// TwinCAT 3 PLC project MOTOR_TESTI
// ProgramVersion: 3.1.4024.0
// libraries:
//   Tc2_ControllerToolbox, * (Beckhoff Automation GmbH)
//   Tc2_EtherCAT, * (Beckhoff Automation GmbH)
//   Tc2_MC2, * (Beckhoff Automation GmbH)
//   Tc2_Standard, * (Beckhoff Automation GmbH)
//   Tc2_System, * (Beckhoff Automation GmbH)
//   Tc3_Module, * (Beckhoff Automation GmbH)
// project tree:
//   GVLs/ MAIN_GVL.TcGVL
//   / PlcTask.TcTTO
//   POUs/ COE_READ_WRITE.TcPOU, MAIN.TcPOU, SINGEN.TcPOU
// real-time tasks:
//   TASK PlcTask: cycle T#10ms, priority 20, ADS port 350
// motion (NC):
//   TASK NC-Task 1 SAF: cycle T#10ms, priority 4, ADS port 501
//   TASK NC-Task 1 SVB: cycle T#10ms, priority 8, ADS port 511
//   AXIS Axis 1 (id 1)
//     General: UnitName=°
//     Velo: Maximum=9600
//     OtherSettings: AllowMotionCmdToSlave=true
//     encoder EncType=19
//       EncPara: ScaleFactorNumerator=0.087890625, MaxCount=#xffffffff
//     drive DrvType=16
//       DrvPara: MaxCount=#xffffffff
//         Analog: VeloReferenz=9600, TorqueSetpointScale=10, ScaleFactorActTorque=0.1
//         TimeComp: TaskDelayCycles=1
//     controller CtrType=1
//       CtrPara: PriorControlFactor=1
//         PosDiffControl: Enable=false
//         Observer: BandWidth=20
// I/O:
//   DEVICE Device 5 (EtherCAT), AmsNetId 192.168.137.220.6.1
//     Term 1 (EK1100) [EK1100 EtherCAT Coupler (2A E-Bus)]
//       Term 2 (EL3004) [EL3004 4Ch. Ana. Input +/-10V]
//       Term 3 (EL3218) [EL3218-0000 8Ch. Ana. Input PT100 (RTD)]
//       Term 4 (EL1809) [EL1809 16Ch. Dig. Input 24V, 3ms]
//       Term 5 (EL2809) [EL2809 16Ch. Dig. Output 24V, 0.5A]
//       Term 7 (EL9011) [EL9011 End Terminal]
//     Drive 6 (
            HiDrive
        ) [HiDrive - EtherCAT (CoE) - Profile: Basic & Object Dictionary (v.7.0)]
// variable links:
//   NC-Task 1 SAF/Axes/Axis 1 <-> Device 5 (EtherCAT)/Drive 6 (
            HiDrive
        )
//     Drive/Inputs/In/nState1 <-> Tx PDO4/Status Word
//     Drive/Inputs/In/nState2 <-> Tx PDO4/Status Word @bit 8
//     Drive/Inputs/In/nState4 @bit 1 <-> WcState/InputToggle
//     Drive/Inputs/In/nState4 <-> WcState/WcState
//     Drive/Outputs/Out/nCtrl1 <-> Rx PDO4/Control Word
//     Drive/Outputs/Out/nCtrl2 <-> Rx PDO4/Control Word @bit 8
//     Enc/Inputs/In/nDataIn1 <-> Tx PDO4/Position Actual Value
//     Enc/Inputs/In/nState4 @bit 1 <-> WcState/InputToggle
//     Enc/Inputs/In/nState4 <-> WcState/WcState
//   MOTOR_TESTI/MOTOR_TESTI Instance <-> Device 5 (EtherCAT)/Drive 6 (
            HiDrive
        )
//     PlcTask Inputs/MAIN.OPERATING_MODE_1_READ <-> Tx PDO3/Pr[181] - Operating Mode
//     PlcTask Inputs/MAIN.TORQUE_MONITOR_1 <-> Tx PDO3/Pr[35] - Torque Monitor [0.1% Ipeak]
//     PlcTask Inputs/MAIN.WINDING_THERMAL_IMAGE <-> Tx PDO3/Pr[36] - Winding Thermal Image [0.1%]
//     PlcTask Outputs/MAIN.HIDRIVE_PLC_OUT_1 <-> Rx PDO4/Target Position
//     PlcTask Outputs/MAIN.OPERATING_MODE_1_WRITE <-> Rx PDO3/Pr[181] - Operating Mode
//     PlcTask Outputs/SINGEN.PR5_INTERNALSETPOINT_1 <-> Rx PDO3/Pr[5] - Internal SetPoint [rpm]
//   MOTOR_TESTI/MOTOR_TESTI Instance <-> Device 5 (EtherCAT)/Term 1 (EK1100)/Term 2 (EL3004)
//     PlcTask Inputs/MAIN.TEST_TORQUE_SENSOR_1 <-> AI Standard Channel 3/Value
//     PlcTask Inputs/MAIN.VOL_READ_1 <-> AI Standard Channel 1/Value
//     PlcTask Inputs/MAIN.VOL_READ_2 <-> AI Standard Channel 2/Value
//   MOTOR_TESTI/MOTOR_TESTI Instance <-> NC-Task 1 SAF/Axes/Axis 1
//     PlcTask Inputs/MAIN.HIDRIVE_PLC_IN_1 <-> Drive/Outputs/Out/nDataOut1
//     PlcTask Inputs/MAIN_GVL.MOTOR_AXIS1.NcToPlc <-> Outputs/ToPlc
//     PlcTask Outputs/MAIN_GVL.MOTOR_AXIS1.PlcToNc <-> Inputs/FromPlc

CONFIGURATION MOTOR_TESTI
    RESOURCE PLC ON TwinCAT3
        TASK PlcTask(INTERVAL := T#10ms, PRIORITY := 20);
        PROGRAM MAIN WITH PlcTask : MAIN;
    END_RESOURCE
END_CONFIGURATION

// ---- GVLs/MAIN_GVL.TcGVL
{attribute 'qualified_only'}
VAR_GLOBAL
	
	MC_POWER_MOTOR: MC_POWER;
	MOTOR_AXIS1: AXIS_REF;
	
	ENABLE_MOTOR: BOOL;
	OverrideRatio: REAL:=100;
END_VAR

// ---- POUs/MAIN.TcPOU
PROGRAM MAIN
VAR
	HIDRIVE_PLC_IN_1 AT%I* : DINT; // MOTION/DRIVE İÇİNDE / OUTPUT / NDATAOUT1 LİNKİNE EKLENİR
	HIDRIVE_PLC_OUT_1 AT%Q* : DINT; // HIDRIVE İÇİNDE RX PDO4 İÇİNDEKİ TARGET POSİTİONA LİNKLENİR BU LİNKLEME YAPILMAZSA MOTOR ÇALIŞMAZ
	TORQUE_MONITOR_1 AT%I* : INT ;
	CURRENT_ACTUAL : REAL;
	MAX_PEEK_CURRENT : INT := 10;
	
	OPERATING_MODE_1_WRITE AT%Q* : INT:=203; // 0 SPEED CONTROL - 203 ETHERCAT - 110 CURRENT
		OPERATING_MODE_1_READ AT%I* : INT; // 0 SPEED CONTROL - 203 ETHERCAT - 110 CURRENT
		OPERATING_MODE_1_READ_SCADA: REAL;
		//ug
		WINDING_THERMAL_IMAGE AT %I* : INT;
	OPMODE_CHANGE: BOOL;
	OPMODE: REAL;
	VOL_READ_1 AT %I* : INT ;
	VOL_READ_2 AT %I* : INT ;
	TORQ_VOLTAGE_HESAP : REAL;
	TORQ_VOLTAGE_OFFSET : REAL := 2.63;
	TORQ_VOLTAGE_FARK : REAL;
	A : LREAL := -3.00499219E-02;
	B : LREAL := 1.73472887E-02;
	C : LREAL := 9.69692536E+00;
	TORQ_ACTUAL : LREAL;
	
	M_TORQ : REAL := 9.2348; // 9.2348
	N_TORQ : REAL := -24.057; // -24.057
	TEST_TORQUE_SENSOR_1 AT %I* : INT ;
	M_TEST : INT := 409;
	N_TEST : INT := 204;
	KISSLER_TORQUE_SENSOR_SCALED: REAL;

	REVOLUTION_RadSn : REAL;
	REVOLUTION_RPM: LREAL; //FROM BECKHOFF NC ( NUMERIC/Motion CONTROL )
	
	Torque_Offset : REAL;
	
	
//	bStartScope : BOOL;
//	bStopScope : BOOL;
//	bExportScope : BOOL;
//	Kontrol1: BOOL;
//	Kontrol2: BOOL;
//	Kontrol3: BOOL;
	
//	SET_TO_SETPOINT2 : INT;
	
//	StartCase: BOOL;
//	RestartCase: BOOL;
	
//	fbTimer: TON;
//	bTriggerTimer1: BOOL;
//	bTriggerTimer2: BOOL;
//	bTriggerTimer3: BOOL;

//	nState: UDINT := 0;
	
	eReqState	:BOOL;
	
END_VAR

REVOLUTION_RPM:=(Main_Gvl.MOTOR_AXIS1.NcToPlc.ActVelo/360)*60;
CURRENT_ACTUAL := INT_TO_REAL(TORQUE_MONITOR_1) * MAX_PEEK_CURRENT / 1000;
IF HIDRIVE_PLC_OUT_1=0 THEN
	MAIN_GVL.ENABLE_MOTOR:=FALSE;
END_IF
HIDRIVE_PLC_OUT_1 := HIDRIVE_PLC_IN_1;
OPERATING_MODE_1_READ_SCADA:=INT_TO_REAL(OPERATING_MODE_1_READ);
IF OPMODE_CHANGE THEN
	OPERATING_MODE_1_WRITE:=REAL_TO_INT(OPMODE);
	OPMODE_CHANGE:=FALSE;
END_IF

//TORQ_HESAP_1 := M_TORQ*((VOL_READ_1/32768)*10) - N_TORQ;
TORQ_VOLTAGE_HESAP := INT_TO_REAL(VOL_READ_1)/32768 *10;

TORQ_VOLTAGE_FARK := TORQ_VOLTAGE_HESAP - TORQ_VOLTAGE_OFFSET;
TORQ_ACTUAL := A*(TORQ_VOLTAGE_FARK*TORQ_VOLTAGE_FARK*TORQ_VOLTAGE_FARK) + B*(TORQ_VOLTAGE_FARK*TORQ_VOLTAGE_FARK) + C*TORQ_VOLTAGE_FARK;


REVOLUTION_RadSn := REVOLUTION_RPM*2*3.14159/60;

KISSLER_TORQUE_SENSOR_SCALED:=((INT_TO_REAL(VOL_READ_1)-8192)/6554)*17.5;

MAIN_GVL.MC_POWER_MOTOR(
	Axis:=MAIN_GVL.MOTOR_AXIS1 , 
	Enable:=MAIN_GVL.ENABLE_MOTOR , 
	Enable_Positive:=MAIN_GVL.ENABLE_MOTOR , 
	Enable_Negative:=MAIN_GVL.ENABLE_MOTOR , 
	Override:=MAIN_GVL.OverrideRatio, 
	BufferMode:= , 
	Options:= , 
	Status=> , 
	Busy=> , 
	Active=> , 
	Error=> , 
	ErrorID=> );
	

	
	
	COE_READ_WRITE();
	SINGEN();

END_PROGRAM

// ---- POUs/COE_READ_WRITE.TcPOU
PROGRAM COE_READ_WRITE
VAR
coe_write          : FB_EcCoESdoWrite; // Function Block for writing in CoE
   coe_read           : FB_EcCoESdoRead;  // Function Block for reading from CoE
   userNetId             : T_AmsNetId := '5.94.222.87.1.1'; // Have to be entered
   userSlaveAddr         : UINT := 1006;     // Have to be entered
   startWrite            : BOOL := FALSE;    // Sign for start writing
   startRead             : BOOL := FALSE;    // Sign for start reading
   nState                : BYTE := 0;        // RW-status
   // Example: Read EL3751 PAI Internal Data: Temperature Value
   int16Buffer           : INT;              // Buffer for reading
   // Example: Select EL3751 Filter1: 22 = IIR Butterw. LP 5th Ord. 1000 Hz:
   uint16Buffer          : UINT:=22;         // Buffer for writing
   bTxPDOState AT%I*     : BOOL;             // (PDO for synchronization)
	EXEC: BOOL;
	bBusy: STRING(INT#4);
	EXEC_wRITE: BOOL;
END_VAR


coe_read(
   sNetId:= '5.94.222.87.1.1', 
   nSlaveAddr:= userSlaveAddr, 
   nSubIndex:= 16#11, 
   nIndex:= 16#2000,
   pDstBuf:= ADR(int16Buffer), 
   cbBufLen:= 16, 
   bExecute:= EXEC, 
   tTimeout:= T#1S,
   );
    // Write entry
   coe_write(
   sNetId:= userNetId,
   nSlaveAddr:= userSlaveAddr,
   nSubIndex:= 16#11,
   nIndex:= 16#2000,
   pSrcBuf:= ADR(uint16Buffer),
   cbBufLen:= 2,
   bExecute:= EXEC_wRITE,
   tTimeout:= T#1S
   );

END_PROGRAM

// ---- POUs/SINGEN.TcPOU
PROGRAM SINGEN
VAR
	DEGREE: INT;
	SINE_MODE_SELECT: REAL;
	SINGEN: FB_CTRL_SIGNAL_GENERATOR;
	SINGEN_SWEEP: FB_CTRL_SIGNAL_GENERATOR;
	State: E_CTRL_STATE;
	ErrorID: E_CTRL_ERRORCODES;
	Error: BOOL;
	WaveOutput: LREAL;
	stParams_deneme: ST_CTRL_SIGNAL_GENERATOR_PARAMS;
	SineSweep_params: ST_CTRL_SIGNAL_GENERATOR_PARAMS;
	Signal_Type: E_CTRL_SIGNAL_TYPE;
	
	SET_TO_SETPOINT: REAL;

	start : BOOL;
	
	eMode_deneme: E_CTRL_MODE;
	SINE_SWEEP: BOOL;
	CLOCK: INT;

	CLOCK_1: INT;
	AT_OFFSET: BOOL;
	SINE_GENERATOR: BOOL;
	
	RPM_TO_Degree_1: LREAL;
	PR5_INTERNALSETPOINT_1 AT%Q*: INT;
	CURRENT_REFERENCE : INT;
	VELOCITY_REFERENCE_rpm : INT;
	VELOCITY_REFERENCE_RadSn : LREAL;
	
	RPM_TO_Degree_2: LREAL;
	PR5_INTERNALSETPOINT_2 AT%Q*: INT;
	
	RPM_TO_Degree_4: LREAL;
	PR5_INTERNALSETPOINT_4 AT%Q*: INT;
	
	RPM_TO_Degree_5: LREAL;
	PR5_INTERNALSETPOINT_5 AT%Q*: INT;
	
	SineWave_PERIOD: TIME:=T#10S;
	SineSweep_PERIOD:TIME:=T#10S;
	MANUAL_SET_POINT: BOOL;
	
	SINE_OFFSET: REAL:=0;
	SINE_AMPLITUDE: REAL:=10;
	CTRL_CYCLE_TIME: TIME:=T#10MS;
	CTRL_TIME_FROM_SCADA: REAL:=10;
	TASK_CYCLE_TIME: TIME:=T#10MS;
	TASK_TIME_FROM_SCADA : REAL:=10;
	PERIOD_FROM_SCADA: REAL:=10;
	
	START_TIME_OFFSET: TIME:=T#0MS;
	START_TIME_FROM_SCADA:REAL;
	
	MAX_SineSweep_PERIOD: TIME := T#1000MS;
	MAX_SineSweep_PERIOD_FROM_SCADA: REAL:=1000;
	SET_SETPOINT_0: BOOL;
	START_SINE: BOOL;
	STOP_SINE: BOOL;
	SCADA_ONLINE: BOOL:=TRUE;
	FB_CTRL_GET_TASK_CYCLETIME: FB_CTRL_GET_TASK_CYCLETIME;
	TaskCycleTime: TIME;
	bCycleTimeValid: BOOL;
	eState: Tc2_ControllerToolbox.E_CTRL_STATE;
	ErrID: Tc2_ControllerToolbox.E_CTRL_ERRORCODES;
	Err: BOOL;
	check1: BOOL;
	FALLDOWN_RATIO: REAL:=2;
	SWEEPPERIOD_FROM_SCADA: REAL;
	ONE_TIME_CHECK: BOOL;
	ONE_TIME_CHECK2: BOOL;
	SinSweep_PERIOD_FOR_SCADA: REAL;
	MAX_SineSweep_PERIOD_FOR_SCADA: REAL;
	START_TIME_OFFSET_FOR_SCADA: REAL;
	TASK_CYCLE_TIME_FOR_SCADA: REAL;
	SineSweep_PERIOD_FOR_SCADA:REAL;
	SineWave_PERIOD_FOR_SCADA:REAL;
	CTRL_CYCLE_TIME_FOR_SCADA:REAL;
	
	torqueValues: ARRAY[0..19] OF REAL := [-150, -120, -100 , -80, -60, -40, -20, -10, -5, -1, 1, 5, 10, 20, 40, 60, 80, 100, 120, 150];
	torqueGain : REAL := 1;
	counter: INT := 0;
	index: INT := 0;
	duration: INT := 500;
	
	bSingenStartScope : BOOL;
	bSingenStopScope : BOOL;
	bSingenExportScope : BOOL;
	
	Kontrol1: BOOL;
	Kontrol2: BOOL;
	Kontrol3: BOOL;
	
	StartCase: BOOL;
	RestartCase: BOOL;
	
	fbTimer1: TON;
	fbTimer2: TON;
	fbTimer3: TON;

	bTriggerTimer1: BOOL;
	bTriggerTimer2: BOOL;
	bTriggerTimer3: BOOL;

	nState: UDINT := 0;
	
END_VAR

CURRENT_REFERENCE := PR5_INTERNALSETPOINT_1;
VELOCITY_REFERENCE_rpm := PR5_INTERNALSETPOINT_1;
VELOCITY_REFERENCE_RadSn := VELOCITY_REFERENCE_rpm*2*3.14159/60;

RPM_TO_Degree_1:= (INT_TO_REAL(PR5_INTERNALSETPOINT_1)/60)*360;
RPM_TO_Degree_2:= (INT_TO_REAL(PR5_INTERNALSETPOINT_2)/60)*360;
RPM_TO_Degree_4:= (INT_TO_REAL(PR5_INTERNALSETPOINT_4)/60)*360;
RPM_TO_Degree_5:= (INT_TO_REAL(PR5_INTERNALSETPOINT_5)/60)*360;


IF counter < duration AND start THEN
	SET_TO_SETPOINT := torqueValues[index]* 9.5493;
	counter := counter + 1;
	IF index > 19 THEN
		SET_TO_SETPOINT := 0;
		index := 0;
		start := FALSE;
	END_IF
	
ELSIF start AND counter >= duration THEN
	index := index +1;
	counter := 0;
END_IF

IF (RestartCase = TRUE) THEN
	nState := 0;	
    bSingenStartScope:=FALSE;
	bSingenStopScope:=FALSE;
	bSingenExportScope:=FALSE;	
	RestartCase := FALSE;
	StartCase := FALSE;
END_IF

CASE nState OF
0:
	IF (StartCase = TRUE) THEN		
		bSingenStartScope:=TRUE;
   	    nState := 10;	
	END_IF

10:
    IF bSingenStartScope THEN
        bTriggerTimer1 := TRUE;
        nState := 20;
    END_IF
20:
    IF (Kontrol1 = TRUE) THEN
        bTriggerTimer1 := FALSE;
		SET_TO_SETPOINT:= 1000;
		PR5_INTERNALSETPOINT_1:=REAL_TO_INT(SET_TO_SETPOINT);
        bTriggerTimer2 := TRUE;
        nState := 30;
    END_IF
30:
    IF (Kontrol2 = TRUE) THEN
        bTriggerTimer2 := FALSE;
		SET_TO_SETPOINT:= 0;
		PR5_INTERNALSETPOINT_1:=REAL_TO_INT(SET_TO_SETPOINT);
        bTriggerTimer3 := TRUE;
        nState := 40;
    END_IF
40: 
    IF (Kontrol3 = TRUE) THEN
        bTriggerTimer3 := FALSE;
		bSingenStopScope := TRUE;
        nState := 50;
    END_IF
50:
    IF bSingenStopScope THEN
        bSingenExportScope:=TRUE;
		//RestartCase := TRUE;

    END_IF
END_CASE

fbTimer1(IN:=bTriggerTimer1, PT:=T#1S, Q=> Kontrol1);	
fbTimer2(IN:=bTriggerTimer2, PT:=T#5S, Q=> Kontrol2);	
fbTimer3(IN:=bTriggerTimer3, PT:=T#1S, Q=> Kontrol3);


IF MANUAL_SET_POINT THEN
	PR5_INTERNALSETPOINT_1:=REAL_TO_INT(SET_TO_SETPOINT);
	PR5_INTERNALSETPOINT_2:=REAL_TO_INT(SET_TO_SETPOINT);
	PR5_INTERNALSETPOINT_4:=REAL_TO_INT(SET_TO_SETPOINT);
	PR5_INTERNALSETPOINT_5:=REAL_TO_INT(SET_TO_SETPOINT);
	IF SET_SETPOINT_0 THEN
	SET_TO_SETPOINT:=0;

	SET_SETPOINT_0:=FALSE;
END_IF



ELSIF NOT MANUAL_SET_POINT AND NOT(SINE_GENERATOR OR SINE_SWEEP) THEN
	PR5_INTERNALSETPOINT_1:=0;
	PR5_INTERNALSETPOINT_2:=0;
	PR5_INTERNALSETPOINT_4:=0;
	PR5_INTERNALSETPOINT_5:=0;
END_IF



IF START_SINE THEN
	eMode_deneme := E_CTRL_MODE.eCTRL_MODE_ACTIVE;
	START_SINE:=FALSE;
	check1:=TRUE;
END_IF

IF STOP_SINE THEN
	eMode_deneme:= e_CTRL_MODE.eCTRL_MODE_PASSIVE;
	STOP_SINE:=FALSE;
END_IF

IF (SINE_GENERATOR AND SINE_SWEEP) OR MANUAL_SET_POINT THEN
	eMode_deneme:=e_CTRL_MODE.eCTRL_MODE_PASSIVE;
END_IF

/// scada tarafından 0 gelirse sinus 1 gelirse saw 2 gelirse triangle
IF SINE_MODE_SELECT=0 THEN
Signal_Type:=E_CTRL_SIGNAL_TYPE.eCTRL_SINUS;
ELSIF SINE_MODE_SELECT=1 THEN
Signal_Type:=E_CTRL_SIGNAL_TYPE.eCTRL_SAWTOOTH;
ELSIF SINE_MODE_SELECT=2 THEN
Signal_Type:=E_CTRL_SIGNAL_TYPE.eCTRL_TRIANGLE;
END_IF

IF SCADA_ONLINE AND NOT (eMode_DENEME= E_CTRL_MODE.eCTRL_MODE_ACTIVE) THEN
CTRL_CYCLE_TIME:=LREAL_TO_TIME(CTRL_TIME_FROM_SCADA);
SineWave_PERIOD:=LREAL_TO_TIME(PERIOD_FROM_SCADA);
SineSweep_PERIOD:=LREAL_TO_TIME(SWEEPPERIOD_FROM_SCADA);
MAX_SineSweep_PERIOD:=REAL_TO_TIME(MAX_SineSweep_PERIOD_FROM_SCADA);
TASK_CYCLE_TIME:=LREAL_TO_TIME(TASK_TIME_FROM_SCADA);
START_TIME_OFFSET:=LREAL_TO_TIME(START_TIME_FROM_SCADA);

END_IF 
IF SINE_GENERATOR THEN
	//SINE Dalgasıın parametreleri, gerekli bilgi infosys de bulunabilir.
	stParams_deneme.eSignalType:=Signal_TYPE;
	stParams_deneme.fAmplitude:=SINE_AMPLITUDE;
	stParams_deneme.tCtrlCycleTime:=CTRL_CYCLE_TIME;
	stParams_deneme.tCylceDuration:=SineWave_PERIOD  ;
	stParams_deneme.tStart:=START_TIME_OFFSET;
	stParams_deneme.tTaskCycleTime:=TASK_CYCLE_TIME;
	stParams_deneme.fOffset:=SINE_OFFSET;
	
	IF eMode_deneme = E_CTRL_MODE.eCTRL_MODE_RESET THEN
		SINGEN(
		fManValue:=, 
		eMode:=eMode_deneme, 
		fOut=> WaveOutput, 
		eState=> State, 
		eErrorId=> ErrorID, 
		bError=> Error, 
		stParams:= SineSweep_params);
	END_IF
	
	IF eMode_deneme = E_CTRL_MODE.eCTRL_MODE_ACTIVE AND AT_OFFSET THEN
		SINGEN(
			fManValue:=, 
			eMode:=eMode_deneme, 
			fOut=> WaveOutput, 
			eState=> State, 
			eErrorId=> ErrorID, 
			bError=> Error, 
			stParams:= stParams_deneme);
		END_IF
		IF eMode_deneme = E_CTRL_MODE.eCTRL_MODE_ACTIVE AND AT_OFFSET THEN
			SET_TO_SETPOINT:=WaveOutput;
			PR5_INTERNALSETPOINT_1:=REAL_TO_INT(SET_TO_SETPOINT);
			PR5_INTERNALSETPOINT_2:=REAL_TO_INT(SET_TO_SETPOINT);
			PR5_INTERNALSETPOINT_4:=REAL_TO_INT(SET_TO_SETPOINT);
			PR5_INTERNALSETPOINT_5:=REAL_TO_INT(SET_TO_SETPOINT);
		END_IF
	END_IF

IF SINE_SWEEP THEN
	//SINE Dalgasıın parametreleri, gerekli bilgi infosys de bulunabilir.
	SineSweep_params.eSignalType:=Signal_TYPE;
	SineSweep_params.fAmplitude:=SINE_AMPLITUDE;
	SineSweep_params.tCtrlCycleTime:=T#10MS;
	SineSweep_params.tCylceDuration:=SineSweep_PERIOD ;
	SineSweep_params.tStart:=T#0MS;
	SineSweep_params.tTaskCycleTime:=T#10MS;
	SineSweep_params.fOffset:=SINE_OFFSET;
	IF eMode_deneme = E_CTRL_MODE.eCTRL_MODE_RESET THEN
		SINGEN_SWEEP(
		fManValue:=, 
		eMode:=eMode_deneme, 
		fOut=> WaveOutput, 
		eState=> State, 
		eErrorId=> ErrorID, 
		bError=> Error, 
		stParams:= SineSweep_params);
	END_IF
	IF eMode_deneme = E_CTRL_MODE.eCTRL_MODE_ACTIVE AND AT_OFFSET THEN
		
		SINGEN_SWEEP(
		fManValue:=, 
		eMode:=eMode_deneme, 
		fOut=> WaveOutput, 
		eState=> State, 
		eErrorId=> ErrorID, 
		bError=> Error, 
		stParams:= SineSweep_params);
		
		IF eMode_deneme = E_CTRL_MODE.eCTRL_MODE_ACTIVE AND AT_OFFSET THEN
			SET_TO_SETPOINT:=LREAL_TO_INT(WaveOutput);
			PR5_INTERNALSETPOINT_1:=REAL_TO_INT(SET_TO_SETPOINT);
			PR5_INTERNALSETPOINT_2:=REAL_TO_INT(SET_TO_SETPOINT);
			PR5_INTERNALSETPOINT_4:=REAL_TO_INT(SET_TO_SETPOINT);
			PR5_INTERNALSETPOINT_5:=REAL_TO_INT(SET_TO_SETPOINT);
		END_IF
		
	END_IF
END_IF

//SINE SWEEP TESTININ GERÇEKLEŞTIRILEBILMESI İÇİN HER SINUS DALGASININ ARDINDAN ÖNCEKININ YARISI PERIYODUNDA
//BIR SINUS DALGASININ YARATILMASINI SAĞLAR,0.5HZ'den daha yüksek HZ de bir dalga yaratılmasını önler
IF SINE_SWEEP THEN
	IF eMode_deneme=E_CTRL_MODE.eCTRL_MODE_ACTIVE AND AT_OFFSET THEN
		CLOCK:=CLOCK+1;
	END_IF
	IF CLOCK/(TIME_TO_INT(SineSweep_params.tCylceDuration)/TIME_TO_INT(SineSweep_params.tCtrlCycleTime))= 1 AND SineSweep_PERIOD > MAX_SineSweep_PERIOD THEN
		SineSweep_PERIOD:=REAL_TO_TIME(TIME_TO_REAL(SineSweep_PERIOD)/FALLDOWN_RATIO);
		CLOCK:=0;
	END_IF
	IF SineSweep_PERIOD < MAX_SineSweep_PERIOD THEN
		eMode_deneme:=e_CTRL_MODE.eCTRL_MODE_PASSIVE;
	END_IF
END_IF

// SINE SWEEP MODUNDA MOTORUN EN BAŞTA VERILEN OFFSET DERECESINE KADEMELI OLARAK ÇIKMASINI SINUS DALGASI DURDURULDUKTAN SONRA DA KADEMELI
//OLARAK 0 DEĞERINE İNMESİNİ SAĞLAR
IF eMode_deneme= e_CTRL_MODE.eCTRL_MODE_PASSIVE AND(SINE_SWEEP OR SINE_GENERATOR) THEN
	
	IF PR5_INTERNALSETPOINT_1 > 0 THEN
		CLOCK_1:=CLOCK_1 + 1 ;
		IF CLOCK_1 MOD 10 = 0 THEN
			PR5_INTERNALSETPOINT_1:=PR5_INTERNALSETPOINT_1-1;
			PR5_INTERNALSETPOINT_2:=PR5_INTERNALSETPOINT_1;
			PR5_INTERNALSETPOINT_4:=PR5_INTERNALSETPOINT_1;
			PR5_INTERNALSETPOINT_5:=PR5_INTERNALSETPOINT_1;
			SET_TO_SETPOINT:=PR5_INTERNALSETPOINT_1;
		END_IF
	ELSIF PR5_INTERNALSETPOINT_1 < 0 THEN
		CLOCK_1:=CLOCK_1 + 1 ;
		IF CLOCK_1 MOD 10 = 0 THEN
			PR5_INTERNALSETPOINT_1:=PR5_INTERNALSETPOINT_1+1;
			PR5_INTERNALSETPOINT_2:=PR5_INTERNALSETPOINT_1;
			PR5_INTERNALSETPOINT_4:=PR5_INTERNALSETPOINT_1;
			PR5_INTERNALSETPOINT_5:=PR5_INTERNALSETPOINT_1;
			SET_TO_SETPOINT:=PR5_INTERNALSETPOINT_1;
			
		END_IF
	ELSIF PR5_INTERNALSETPOINT_1=0 THEN
		CLOCK_1:=0;
		AT_OFFSET:=FALSE;
		eMode_deneme:=e_cTRL_MODE.eCTRL_MODE_RESET;
	END_IF
	
ELSIF eMode_deneme=e_CTRL_MODE.eCTRL_MODE_ACTIVE AND NOT AT_OFFSET AND (SINE_SWEEP OR SINE_GENERATOR) THEN
	IF PR5_INTERNALSETPOINT_1 > SINE_OFFSET THEN
		CLOCK_1:=CLOCK_1 + 1 ;
		IF CLOCK_1 MOD 10 = 0 THEN
			PR5_INTERNALSETPOINT_1:=PR5_INTERNALSETPOINT_1-1;
			PR5_INTERNALSETPOINT_2:=PR5_INTERNALSETPOINT_1;
			PR5_INTERNALSETPOINT_4:=PR5_INTERNALSETPOINT_1;
			PR5_INTERNALSETPOINT_5:=PR5_INTERNALSETPOINT_1;
			SET_TO_SETPOINT:=PR5_INTERNALSETPOINT_1;
		END_IF
ELSIF PR5_INTERNALSETPOINT_1 < SINE_OFFSET THEN
		CLOCK_1:=CLOCK_1 + 1 ;
		IF CLOCK_1 MOD 10 = 0 THEN
			PR5_INTERNALSETPOINT_1:=PR5_INTERNALSETPOINT_1+1;
			PR5_INTERNALSETPOINT_2:=PR5_INTERNALSETPOINT_1;
			PR5_INTERNALSETPOINT_4:=PR5_INTERNALSETPOINT_1;
			PR5_INTERNALSETPOINT_5:=PR5_INTERNALSETPOINT_1;
			SET_TO_SETPOINT:=PR5_INTERNALSETPOINT_1;
		END_IF
ELSIF PR5_INTERNALSETPOINT_1=SINE_OFFSET THEN
		CLOCK_1:=0;
		AT_OFFSET:=TRUE;
	END_IF
END_IF

SinSweep_PERIOD_FOR_SCADA:=TIME_TO_REAL(SineSweep_PERIOD);
CTRL_CYCLE_TIME_FOR_SCADA:=TIME_TO_REAL(CTRL_CYCLE_TIME);
SineWave_PERIOD_FOR_SCADA:=TIME_TO_REAL(SineWave_PERIOD);
SineSweep_PERIOD_FOR_SCADA:=TIME_TO_REAL(SineSweep_PERIOD);
MAX_SineSweep_PERIOD_FOR_SCADA:=TIME_TO_REAL(MAX_SineSweep_PERIOD);
TASK_CYCLE_TIME_FOR_SCADA:=TIME_TO_REAL(TASK_CYCLE_TIME);
START_TIME_OFFSET_FOR_SCADA:=TIME_TO_REAL(START_TIME_OFFSET);

END_PROGRAM
